INTERFACE ITaskStatus

METHOD Abort
END_METHOD

PROPERTY Busy : BOOL
GET
END_GET
END_PROPERTY

PROPERTY Done : BOOL
GET
END_GET
END_PROPERTY

PROPERTY Error : BOOL
GET
END_GET
END_PROPERTY

END_INTERFACE

(* stored: Version 1.1.0.1, ProductVersion 3.1.4024.4
   Itf ITaskStatus: Id {7d150626-9f01-44ae-8ba9-084d89c9c921}
   Method Abort: Id {0f1fb7b5-4654-4007-bf46-d2949d5415d2}
   Property Busy: Id {5a1b8be5-fd5d-4d07-82d9-bb1a80a942f3}
   Get Get: Id {70d294ee-48c2-49be-a8ab-a055401aff50}
   Property Done: Id {94b70fd2-8935-4c13-a21b-75c9111f8e97}
   Get Get: Id {840a9685-615a-4413-94b3-b12503c1c945}
   Property Error: Id {722230f9-5175-42e5-937e-3a31938fd53a}
   Get Get: Id {f7520206-3d53-4852-8b1f-87aa0a44b267} *)
